// SIMATIC S7-200 SMART project (STEP 7-Micro/WIN SMART), CPU ST60

SYMBOL_TABLE 系统符号
Always_On        SM0.0    // 始终接通
First_Scan_On    SM0.1    // 仅在第一个扫描周期时接通
HSC0_Ctrl        SMB37    // 组态和控制 HSC0
HSC0_CV          SMD38    // HSC0 新当前值
HSC0_PV          SMD42    // HSC0 新预设值
END_SYMBOL_TABLE

ORGANIZATION_BLOCK MAIN:OB1
TITLE=程序注释
BEGIN
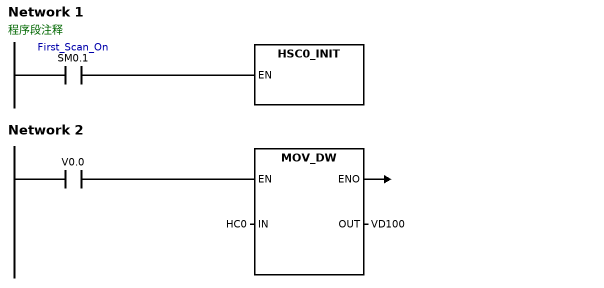
Network 1
// 程序段注释
LD     First_Scan_On:SM0.1
CALL   HSC0_INIT:SBR1
Network 2
LD     V0.0
MOVD   HC0, VD100
END_ORGANIZATION_BLOCK

SUBROUTINE_BLOCK HSC0_INIT:SBR1
TITLE=
BEGIN
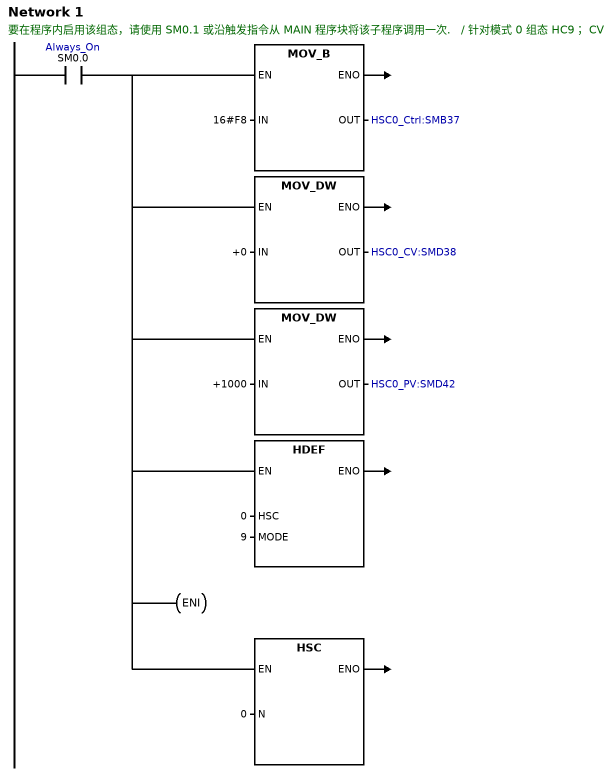
Network 1
// 要在程序内启用该组态，请使用 SM0.1 或沿触发指令从 MAIN 程序块将该子程序调用一次.  
// 针对模式 0 组态 HC9； CV = 0； PV = 1000； 加计数； 
// 启用中断并启动计数器.
// 
//置位控制位： 加计数； 速率 4X； 已启用； 
//装载 CV
//装载 PV
LD     Always_On:SM0.0
MOVB   16#F8, HSC0_Ctrl:SMB37
MOVD   +0, HSC0_CV:SMD38
MOVD   +1000, HSC0_PV:SMD42
HDEF   0, 9
ENI
HSC    0
END_SUBROUTINE_BLOCK
